(* PLC project 04_comparison.project, CODESYS CODESYS V3.5 SP22 Patch 2 *)
(* stored: creationDateTime 2026-07-23T20:19:07.788747, modificationDateTime 2026-07-23T20:18:43.5444979 *)

PROGRAM PLC_PRG
  VAR
    rValue : REAL;
    rLimit : REAL;
    xEnable : BOOL;
    xAlarm : BOOL;
    xGreater : BOOL;
  END_VAR

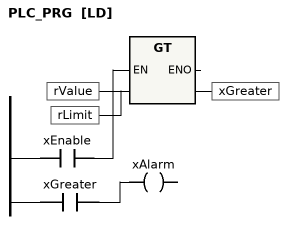
(* LD diagram, written out as Structured Text *)

IF xEnable THEN xGreater := rValue > rLimit; END_IF;

xAlarm := xGreater;
END_PROGRAM

CONFIGURATION Application
  RESOURCE Application ON PLC
    TASK MainTask(INTERVAL := T#20ms, PRIORITY := 1);
    PROGRAM PLC_PRG WITH MainTask : PLC_PRG;
  END_RESOURCE
END_CONFIGURATION
